TYPE Mat53 : ARRAY[1..5, 1..3] OF LREAL; END_TYPE

(* stored: Version 1.1.0.1, ProductVersion 3.1.4024.11
   DUT Mat53: Id {77f2db4c-a423-4a36-b7c6-22368b8a8b7a} *)
